INTERFACE ITF_BaseGroupElement

END_INTERFACE

(* stored: Version 1.1.0.1
   Itf ITF_BaseGroupElement: Id {d28f4434-f18e-0ace-07d5-b8e3255289a2} *)
